FUNCTION_BLOCK WagoInputBlock (* Basic Function Block Type *)
  (* Standard: 61499-2 *)
  (* Version 0.0, 2009-11-20, JHC, University of Auckland *)
  (* Compiler header: package fb.rt.wago; #include "kbusapi.h" *)
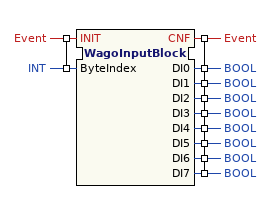
  EVENT_INPUT
    INIT WITH ByteIndex; (* Initialization Request *)
  END_EVENT
  EVENT_OUTPUT
    CNF WITH DI0, DI1, DI2, DI3, DI4, DI5, DI6, DI7; (* Execution Confirmation *)
  END_EVENT
  VAR_INPUT
    ByteIndex : INT;
  END_VAR
  VAR_OUTPUT
    DI0 : BOOL := false;
    DI1 : BOOL := false;
    DI2 : BOOL := false;
    DI3 : BOOL := false;
    DI4 : BOOL := false;
    DI5 : BOOL := false;
    DI6 : BOOL := false;
    DI7 : BOOL := false;
  END_VAR
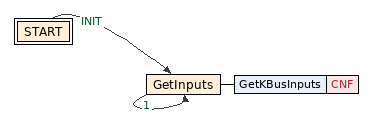
  EC_STATES
    START; (* Initial State *)
    GetInputs : GetKBusInputs -> CNF;
  END_STATES
  EC_TRANSITIONS
    START TO GetInputs := INIT;
    GetInputs TO GetInputs := 1;
  END_TRANSITIONS
  ALGORITHM GetKBusInputs IN Java: (* Normally executed algorithm *)
// read byte from pab and show it on console
KbusOpen();
// read input value
KbusUpdate();

me->DI0 = (0x1 & pstPabIN->uc.Pab[me->ByteIndex]) > 0;
me->DI1 = (0x2 & pstPabIN->uc.Pab[me->ByteIndex]) > 0;
me->DI2 = (0x4 & pstPabIN->uc.Pab[me->ByteIndex]) > 0;
me->DI3 = (0x8 & pstPabIN->uc.Pab[me->ByteIndex]) > 0;
me->DI4 = (0x10 & pstPabIN->uc.Pab[me->ByteIndex]) > 0;
me->DI5 = (0x20 & pstPabIN->uc.Pab[me->ByteIndex]) > 0;
me->DI6 = (0x40 & pstPabIN->uc.Pab[me->ByteIndex]) > 0;
me->DI7 = (0x80 & pstPabIN->uc.Pab[me->ByteIndex]) > 0;

// Close
KbusClose();
  END_ALGORITHM
END_FUNCTION_BLOCK
